FUNCTION_BLOCK FB_RingBufferTests EXTENDS TcUnit.FB_TestSuite
VAR
END_VAR

ConfigureRejectsZeroCapacity();
EmptyAfterConfigure();
PushPopFifoLreal();
PushPopFifoInt();
PushPopUserDefinedStruct();
PeekDoesNotConsume();
WrapAroundPreservesOrder();
PushReturnsFalseWhenFull();
PopReturnsFalseWhenEmpty();

METHOD ConfigureRejectsZeroCapacity : BOOL
VAR
    rb       : T3TckitUtils_Plc.FB_RingBuffer;
    storage  : ARRAY[1..4] OF LREAL;
END_VAR
IF TEST_ORDERED(__POUNAME()) THEN
    AssertFalse(Condition := rb.Configure(storage, 0),
        Message := 'Configure with capacity=0 must return FALSE');
    AssertTrue(Condition := rb.Configure(storage, 4),
        Message := 'Configure with matched diSize/capacity must return TRUE');
    TEST_FINISHED();
END_IF
END_METHOD

METHOD EmptyAfterConfigure : BOOL
VAR
    rb       : T3TckitUtils_Plc.FB_RingBuffer;
    storage  : ARRAY[1..4] OF LREAL;
END_VAR
IF TEST_ORDERED(__POUNAME()) THEN
    AssertTrue(Condition := rb.Configure(storage, 4),
        Message := 'Configure must succeed for ARRAY[1..4] OF LREAL with capacity=4');
    AssertEquals_UDINT(Expected := 0, Actual := rb.Count,
        Message := 'Fresh buffer Count must be 0');
    AssertTrue(Condition := rb.IsEmpty,
        Message := 'Fresh buffer IsEmpty must be TRUE');
    AssertFalse(Condition := rb.IsFull,
        Message := 'Fresh buffer IsFull must be FALSE');
    AssertEquals_UDINT(Expected := 4, Actual := rb.Capacity,
        Message := 'Capacity must reflect the configured value');
    TEST_FINISHED();
END_IF
END_METHOD

METHOD PeekDoesNotConsume : BOOL
VAR
    rb       : T3TckitUtils_Plc.FB_RingBuffer;
    storage  : ARRAY[1..4] OF LREAL;
    v1       : LREAL;
    seen     : LREAL;
END_VAR
IF TEST_ORDERED(__POUNAME()) THEN
    rb.Configure(storage, 4);
    v1 := 7.5;
    rb.Push(v1);
    AssertTrue(Condition := rb.Peek(seen),
        Message := 'Peek must succeed when buffer is non-empty');
    AssertEquals_LREAL(Expected := 7.5, Actual := seen, Delta := 1E-9,
        Message := 'Peek must return the front element');
    AssertEquals_UDINT(Expected := 1, Actual := rb.Count,
        Message := 'Peek must not change Count');
    seen := 0.0;
    rb.Peek(seen);
    AssertEquals_LREAL(Expected := 7.5, Actual := seen, Delta := 1E-9,
        Message := 'A second Peek must return the same element');
    TEST_FINISHED();
END_IF
END_METHOD

METHOD PopReturnsFalseWhenEmpty : BOOL
VAR
    rb       : T3TckitUtils_Plc.FB_RingBuffer;
    storage  : ARRAY[1..4] OF LREAL;
    popped   : LREAL;
END_VAR
IF TEST_ORDERED(__POUNAME()) THEN
    rb.Configure(storage, 4);
    AssertFalse(Condition := rb.Pop(popped),
        Message := 'Pop must return FALSE on an empty buffer');
    AssertFalse(Condition := rb.Peek(popped),
        Message := 'Peek must return FALSE on an empty buffer');
    TEST_FINISHED();
END_IF
END_METHOD

METHOD PushPopFifoInt : BOOL
VAR
    rb       : T3TckitUtils_Plc.FB_RingBuffer;
    storage  : ARRAY[1..4] OF INT;
    v1, v2   : INT;
    popped   : INT;
END_VAR
IF TEST_ORDERED(__POUNAME()) THEN
    rb.Configure(storage, 4);
    v1 := 11;
    v2 := 22;
    rb.Push(v1);
    rb.Push(v2);
    AssertEquals_UDINT(Expected := 2, Actual := rb.Count,
        Message := 'Count after two INT pushes must be 2');
    rb.Pop(popped);
    AssertEquals_INT(Expected := 11, Actual := popped,
        Message := 'INT FIFO order must match LREAL FIFO order');
    rb.Pop(popped);
    AssertEquals_INT(Expected := 22, Actual := popped,
        Message := 'Second INT Pop must return the second Push');
    TEST_FINISHED();
END_IF
END_METHOD

METHOD PushPopFifoLreal : BOOL
VAR
    rb       : T3TckitUtils_Plc.FB_RingBuffer;
    storage  : ARRAY[1..4] OF LREAL;
    v1, v2, v3 : LREAL;
    popped   : LREAL;
END_VAR
IF TEST_ORDERED(__POUNAME()) THEN
    rb.Configure(storage, 4);
    v1 := 1.0;
    v2 := 2.0;
    v3 := 3.0;
    AssertTrue(Condition := rb.Push(v1), Message := 'Push(1.0) must succeed');
    AssertTrue(Condition := rb.Push(v2), Message := 'Push(2.0) must succeed');
    AssertTrue(Condition := rb.Push(v3), Message := 'Push(3.0) must succeed');
    AssertEquals_UDINT(Expected := 3, Actual := rb.Count,
        Message := 'Count after three pushes must be 3');
    AssertTrue(Condition := rb.Pop(popped), Message := 'Pop must succeed when buffer is non-empty');
    AssertEquals_LREAL(Expected := 1.0, Actual := popped, Delta := 1E-9,
        Message := 'First Pop must return the first Push');
    rb.Pop(popped);
    AssertEquals_LREAL(Expected := 2.0, Actual := popped, Delta := 1E-9,
        Message := 'Second Pop must return the second Push');
    rb.Pop(popped);
    AssertEquals_LREAL(Expected := 3.0, Actual := popped, Delta := 1E-9,
        Message := 'Third Pop must return the third Push');
    AssertTrue(Condition := rb.IsEmpty,
        Message := 'Buffer must be empty after popping all elements');
    TEST_FINISHED();
END_IF
END_METHOD

METHOD PushPopUserDefinedStruct : BOOL
VAR
    rb       : T3TckitUtils_Plc.FB_RingBuffer;
    storage  : ARRAY[1..4] OF ST_Sample;
    inA, inB : ST_Sample;
    popped   : ST_Sample;
END_VAR
IF TEST_ORDERED(__POUNAME()) THEN
    rb.Configure(storage, 4);
    inA.t := 0.1; inA.v := 11.0;
    inB.t := 0.2; inB.v := 22.0;
    rb.Push(inA);
    rb.Push(inB);
    AssertEquals_UDINT(Expected := 2, Actual := rb.Count,
        Message := 'Count after two ST_Sample pushes must be 2');
    rb.Pop(popped);
    AssertEquals_LREAL(Expected := 0.1, Actual := popped.t, Delta := 1E-9,
        Message := 'ST_Sample.t must round-trip exactly');
    AssertEquals_LREAL(Expected := 11.0, Actual := popped.v, Delta := 1E-9,
        Message := 'ST_Sample.v must round-trip exactly');
    rb.Pop(popped);
    AssertEquals_LREAL(Expected := 0.2, Actual := popped.t, Delta := 1E-9,
        Message := 'Second ST_Sample.t must round-trip exactly');
    AssertEquals_LREAL(Expected := 22.0, Actual := popped.v, Delta := 1E-9,
        Message := 'Second ST_Sample.v must round-trip exactly');
    TEST_FINISHED();
END_IF
END_METHOD

METHOD PushReturnsFalseWhenFull : BOOL
VAR
    rb       : T3TckitUtils_Plc.FB_RingBuffer;
    storage  : ARRAY[1..2] OF LREAL;
    v1, v2, v3 : LREAL;
END_VAR
IF TEST_ORDERED(__POUNAME()) THEN
    rb.Configure(storage, 2);
    v1 := 1.0; v2 := 2.0; v3 := 3.0;
    AssertTrue(Condition := rb.Push(v1), Message := 'First Push must succeed');
    AssertTrue(Condition := rb.Push(v2), Message := 'Second Push must succeed');
    AssertTrue(Condition := rb.IsFull,
        Message := 'IsFull must be TRUE when Count = Capacity');
    AssertFalse(Condition := rb.Push(v3),
        Message := 'Push must return FALSE when the buffer is full');
    AssertEquals_UDINT(Expected := 2, Actual := rb.Count,
        Message := 'A refused Push must not change Count');
    TEST_FINISHED();
END_IF
END_METHOD

METHOD WrapAroundPreservesOrder : BOOL
VAR
    rb       : T3TckitUtils_Plc.FB_RingBuffer;
    storage  : ARRAY[1..3] OF LREAL;
    a, b, c, d, e : LREAL;
    popped   : LREAL;
END_VAR
IF TEST_ORDERED(__POUNAME()) THEN
    rb.Configure(storage, 3);
    a := 1.0; b := 2.0; c := 3.0;
    rb.Push(a); rb.Push(b); rb.Push(c);
    rb.Pop(popped);
    AssertEquals_LREAL(Expected := 1.0, Actual := popped, Delta := 1E-9,
        Message := 'First Pop must return 1.0 before wrap');
    rb.Pop(popped);
    AssertEquals_LREAL(Expected := 2.0, Actual := popped, Delta := 1E-9,
        Message := 'Second Pop must return 2.0 before wrap');
    d := 4.0; e := 5.0;
    AssertTrue(Condition := rb.Push(d),
        Message := 'Push after Pops must succeed (forces write index to wrap)');
    AssertTrue(Condition := rb.Push(e),
        Message := 'Second Push after Pops must also succeed');
    rb.Pop(popped);
    AssertEquals_LREAL(Expected := 3.0, Actual := popped, Delta := 1E-9,
        Message := 'After wrap, Pop must return 3.0 (the surviving pre-wrap element)');
    rb.Pop(popped);
    AssertEquals_LREAL(Expected := 4.0, Actual := popped, Delta := 1E-9,
        Message := 'After wrap, second Pop must return 4.0');
    rb.Pop(popped);
    AssertEquals_LREAL(Expected := 5.0, Actual := popped, Delta := 1E-9,
        Message := 'After wrap, third Pop must return 5.0');
    TEST_FINISHED();
END_IF
END_METHOD

END_FUNCTION_BLOCK

(* stored: Version 1.1.0.1
   POU FB_RingBufferTests: Id {36ff8f11-bd15-4880-a23d-88dee1f36a1f}, SpecialFunc None
   Method ConfigureRejectsZeroCapacity: Id {6cc22601-6cf8-4382-a0cc-2c88d7983104}
   Method EmptyAfterConfigure: Id {dda7a3e4-275f-4912-95a0-aaba25b2a853}
   Method PeekDoesNotConsume: Id {fa1666d0-e33b-46b1-b1df-0feb03d7462d}
   Method PopReturnsFalseWhenEmpty: Id {faf38b56-7be6-4932-9aaf-6552a54849d3}
   Method PushPopFifoInt: Id {909bce4b-2f7d-4621-a807-3a71dde72646}
   Method PushPopFifoLreal: Id {cc5b4025-a1d1-41ad-8230-6b3272e524e6}
   Method PushPopUserDefinedStruct: Id {19ee25fe-91c5-4a04-b46d-956f98267fcc}
   Method PushReturnsFalseWhenFull: Id {ac9fed72-71ec-4683-bb6b-75c278ad573b}
   Method WrapAroundPreservesOrder: Id {13813ffa-b3b0-48ac-9204-66404483052a} *)
